// TIA Portal V16 export
// export: Created 2026-06-22T07:42:12.1971695Z, ExportSetting WithDefaults, DisplayName Totally Integrated Automation Portal, DisplayVersion V16 Update 8, DisplayName TIA Portal Version Control Interface, DisplayVersion V16 Update 8, DisplayName TIA Portal Openness, DisplayVersion V16 Update 8, DisplayName SINAMICS Startdrive Advanced, DisplayVersion V16, DisplayName SINAMICS Startdrive G130, G150, S120, S150, SINAMICS MV, S210, DisplayVersion V16, DisplayName SINAMICS Startdrive G110M, G120, G120C, G120D, G120P, DisplayVersion V16, DisplayName STEP 7 Professional, DisplayVersion V16 Update 8, DisplayName STEP 7 Safety, DisplayVersion V16 Update 7, DisplayName WinCC Advanced, DisplayVersion V16 Update 8
Screen "Elevator_Monitor"  800x480, Number=1
  ScreenLayer 
    Circle "LMP_Running" at 120,100 size 48x48
      RangeAppearanceAnimation "RangeAppearanceAnimation"
        tag STS_Elevator_Running
        0..0: back #dedbde, fore #181c31
        1..1: back #00ff00, fore #181c31
    Circle "LMP_Fault" at 632,100 size 48x48
      RangeAppearanceAnimation "RangeAppearanceAnimation"
        tag LMP_Elevator_Fault
        0..0: back #dedbde, fore #181c31
        1..1: back #00ff00, fore #181c31
    Circle "LMP_Down" at 504,100 size 48x48
      RangeAppearanceAnimation "RangeAppearanceAnimation"
        tag STS_Elevator_Down
        0..0: back #dedbde, fore #181c31
        1..1: back #00ff00, fore #181c31
    Circle "LMP_Up" at 376,100 size 48x48
      RangeAppearanceAnimation "RangeAppearanceAnimation"
        tag STS_Elevator_Up
        0..0: back #dedbde, fore #181c31
        1..1: back #00ff00, fore #181c31
    Circle "LMP_DoorOpen" at 248,100 size 48x48
      RangeAppearanceAnimation "RangeAppearanceAnimation"
        tag STS_Elevator_DoorOpen
        0..0: back #dedbde, fore #181c31
        1..1: back #00ff00, fore #181c31
    Button "BTN_UpCall" at 135,350 size 130x56  Mode=Text, TextOff="上行呼叫", TextOn="上行呼叫"
      on Press: SetBit(Tag := BTN_Elevator_Up)
      on Release: ResetBit(Tag := BTN_Elevator_Up)
    Button "BTN_EmergencyStop" at 535,350 size 130x56  Mode=Text, TextOff="急停", TextOn="急停"
      on Press: SetBit(Tag := MEM_Elevator_EmergencyStop)
      on Release: ResetBit(Tag := MEM_Elevator_EmergencyStop)
    Button "BTN_DownCall" at 335,350 size 130x56  Mode=Text, TextOff="下行呼叫", TextOn="下行呼叫"
      on Press: SetBit(Tag := BTN_Elevator_Down)
      on Release: ResetBit(Tag := BTN_Elevator_Down)
    IOField "IO_Floor" at 280,200 size 160x70  DataFormat=Decimal, FormatPattern=s99999, Mode=InOutput
      ProcessValue := IO_Elevator_Floor
    TextField "TXT_Title" at 200,25 size 400x40  Text="电梯监控画面"
    TextField "TXT_Floor_Unit" at 450,225 size 40x40  Text="楼"
